// TIA Portal V20 export
TYPE "typeSafetyForcedDoorOpen"
// stored: Access Published, IsFailsafeCompliant true, Namespace Safety
   STRUCT
      Door1OpenMemo : Bool;
      Door2OpenMemo : Bool;
      Door3OpenMemo : Bool;
      Door4OpenMemo : Bool;
      Door5OpenMemo : Bool;
      Door6OpenMemo : Bool;
      Door7OpenMemo : Bool;
      Door1ForcedOpenError : Bool;   // Forced Open UNWIND REAR DOOR
      Door2ForcedOpenError : Bool;   // Forced Open AUTO SPLICE DOOR
      Door3ForcedOpenError : Bool;   // Forced Open UNWIND MAIN DOOR
      Door4ForcedOpenError : Bool;   // Forced Open UNWIND TOP DOOR
      Door5ForcedOpenError : Bool;   // Forced Open UNWIND BTM DOOR
      Door6ForcedOpenError : Bool;   // Forced Open STACK TABLE DOOR
      Door7ForcedOpenError : Bool;   // Forced Open JR WINDER DOOR
      Door1OpenTimeOver : Bool;   // Time Over Open UNWIND REAR DOOR
      Door2OpenTimeOver : Bool;   // Time Over Open AUTO SPLICE DOOR
      Door3OpenTimeOver : Bool;   // Time Over Open UNWIND MAIN DOOR
      Door4OpenTimeOver : Bool;   // Time Over Open UNWIND TOP DOOR
      Door5OpenTimeOver : Bool;   // Time Over Open UNWIND BTM DOOR
      Door6OpenTimeOver : Bool;   // Time Over Open STACK TABLE DOOR
      Door7OpenTimeOver : Bool;   // Time Over Open JR WINDER DOOR
      Door1CloseTimeOver : Bool;   // Time Over Close UNWIND REAR DOOR
      Door2CloseTimeOver : Bool;   // Time Over Close AUTO SPLICE DOOR
      Door3CloseTimeOver : Bool;   // Time Over Close UNWIND MAIN DOOR
      Door4CloseTimeOver : Bool;   // Time Over Close UNWIND TOP DOOR
      Door5CloseTimeOver : Bool;   // Time Over Close UNWIND BTM DOOR
      Door6CloseTimeOver : Bool;   // Time Over Close STACK TABLE DOOR
      Door7CloseTimeOver : Bool;   // Time Over Close JR WINDER DOOR
   END_STRUCT;
END_TYPE
